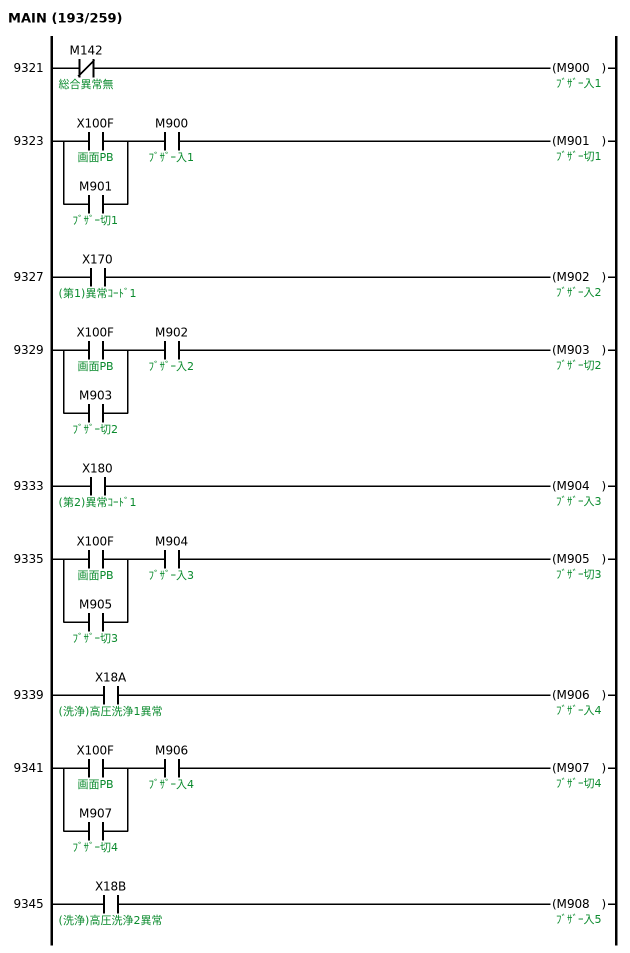
[picture p192: ladder of MAIN, rungs at steps 9321 to 9345]
9321  LDI     M142  ; 総合異常無
      OUT     M900  ; ﾌﾞｻﾞｰ入1
9323  LD      X100F  ; 画面PB
      OR      M901  ; ﾌﾞｻﾞｰ切1
      AND     M900  ; ﾌﾞｻﾞｰ入1
      OUT     M901  ; ﾌﾞｻﾞｰ切1
9327  LD      X170  ; (第1)異常ｺｰﾄﾞ1
      OUT     M902  ; ﾌﾞｻﾞｰ入2
9329  LD      X100F  ; 画面PB
      OR      M903  ; ﾌﾞｻﾞｰ切2
      AND     M902  ; ﾌﾞｻﾞｰ入2
      OUT     M903  ; ﾌﾞｻﾞｰ切2
9333  LD      X180  ; (第2)異常ｺｰﾄﾞ1
      OUT     M904  ; ﾌﾞｻﾞｰ入3
9335  LD      X100F  ; 画面PB
      OR      M905  ; ﾌﾞｻﾞｰ切3
      AND     M904  ; ﾌﾞｻﾞｰ入3
      OUT     M905  ; ﾌﾞｻﾞｰ切3
9339  LD      X18A  ; (洗浄)高圧洗浄1異常
      OUT     M906  ; ﾌﾞｻﾞｰ入4
9341  LD      X100F  ; 画面PB
      OR      M907  ; ﾌﾞｻﾞｰ切4
      AND     M906  ; ﾌﾞｻﾞｰ入4
      OUT     M907  ; ﾌﾞｻﾞｰ切4
9345  LD      X18B  ; (洗浄)高圧洗浄2異常
      OUT     M908  ; ﾌﾞｻﾞｰ入5
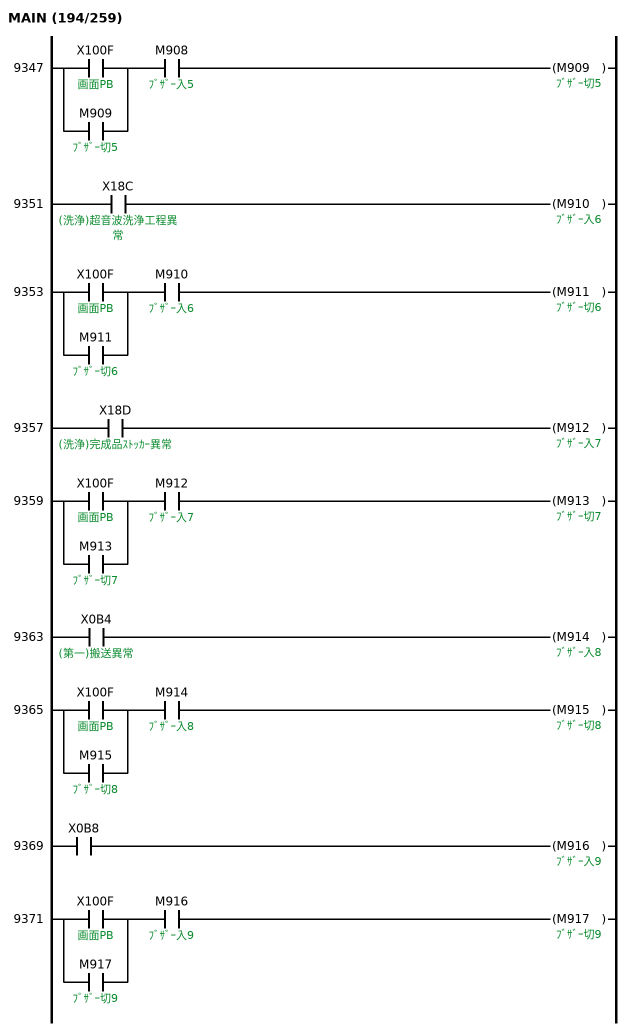
9347  LD      X100F  ; 画面PB
      OR      M909  ; ﾌﾞｻﾞｰ切5
      AND     M908  ; ﾌﾞｻﾞｰ入5
      OUT     M909  ; ﾌﾞｻﾞｰ切5
9351  LD      X18C  ; (洗浄)超音波洗浄工程異常
      OUT     M910  ; ﾌﾞｻﾞｰ入6
9353  LD      X100F  ; 画面PB
      OR      M911  ; ﾌﾞｻﾞｰ切6
      AND     M910  ; ﾌﾞｻﾞｰ入6
      OUT     M911  ; ﾌﾞｻﾞｰ切6
9357  LD      X18D  ; (洗浄)完成品ｽﾄｯｶｰ異常
      OUT     M912  ; ﾌﾞｻﾞｰ入7
9359  LD      X100F  ; 画面PB
      OR      M913  ; ﾌﾞｻﾞｰ切7
      AND     M912  ; ﾌﾞｻﾞｰ入7
      OUT     M913  ; ﾌﾞｻﾞｰ切7
9363  LD      X0B4  ; (第一)搬送異常
      OUT     M914  ; ﾌﾞｻﾞｰ入8
9365  LD      X100F  ; 画面PB
      OR      M915  ; ﾌﾞｻﾞｰ切8
      AND     M914  ; ﾌﾞｻﾞｰ入8
      OUT     M915  ; ﾌﾞｻﾞｰ切8
9369  LD      X0B8
      OUT     M916  ; ﾌﾞｻﾞｰ入9
9371  LD      X100F  ; 画面PB
      OR      M917  ; ﾌﾞｻﾞｰ切9
      AND     M916  ; ﾌﾞｻﾞｰ入9
      OUT     M917  ; ﾌﾞｻﾞｰ切9
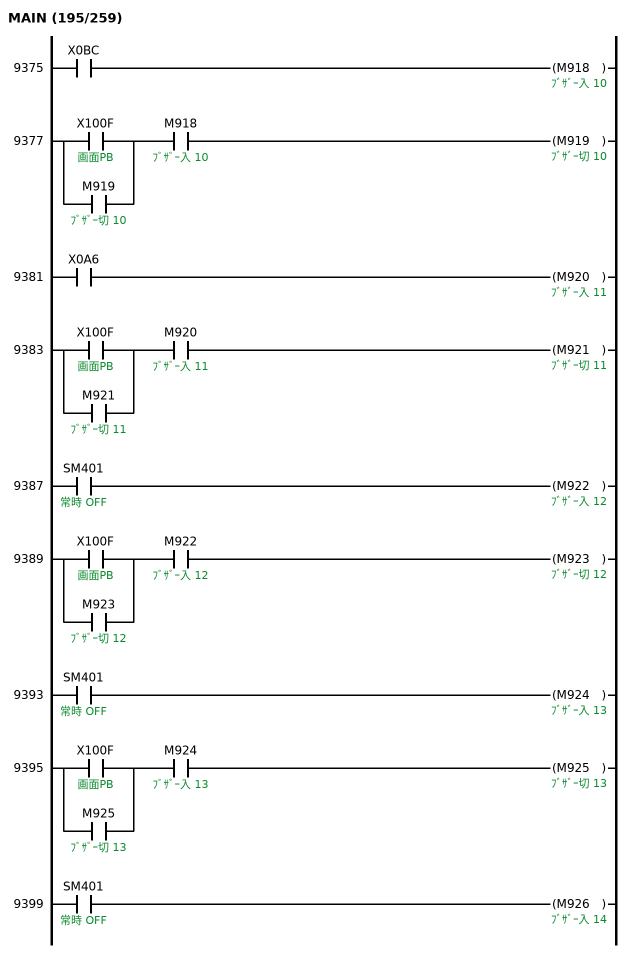
9375  LD      X0BC
      OUT     M918  ; ﾌﾞｻﾞｰ入 10
9377  LD      X100F  ; 画面PB
      OR      M919  ; ﾌﾞｻﾞｰ切 10
      AND     M918  ; ﾌﾞｻﾞｰ入 10
      OUT     M919  ; ﾌﾞｻﾞｰ切 10
9381  LD      X0A6
      OUT     M920  ; ﾌﾞｻﾞｰ入 11
9383  LD      X100F  ; 画面PB
      OR      M921  ; ﾌﾞｻﾞｰ切 11
      AND     M920  ; ﾌﾞｻﾞｰ入 11
      OUT     M921  ; ﾌﾞｻﾞｰ切 11
9387  LD      SM401  ; 常時 OFF
      OUT     M922  ; ﾌﾞｻﾞｰ入 12
9389  LD      X100F  ; 画面PB
      OR      M923  ; ﾌﾞｻﾞｰ切 12
      AND     M922  ; ﾌﾞｻﾞｰ入 12
      OUT     M923  ; ﾌﾞｻﾞｰ切 12
9393  LD      SM401  ; 常時 OFF
      OUT     M924  ; ﾌﾞｻﾞｰ入 13
9395  LD      X100F  ; 画面PB
      OR      M925  ; ﾌﾞｻﾞｰ切 13
      AND     M924  ; ﾌﾞｻﾞｰ入 13
      OUT     M925  ; ﾌﾞｻﾞｰ切 13
9399  LD      SM401  ; 常時 OFF
      OUT     M926  ; ﾌﾞｻﾞｰ入 14
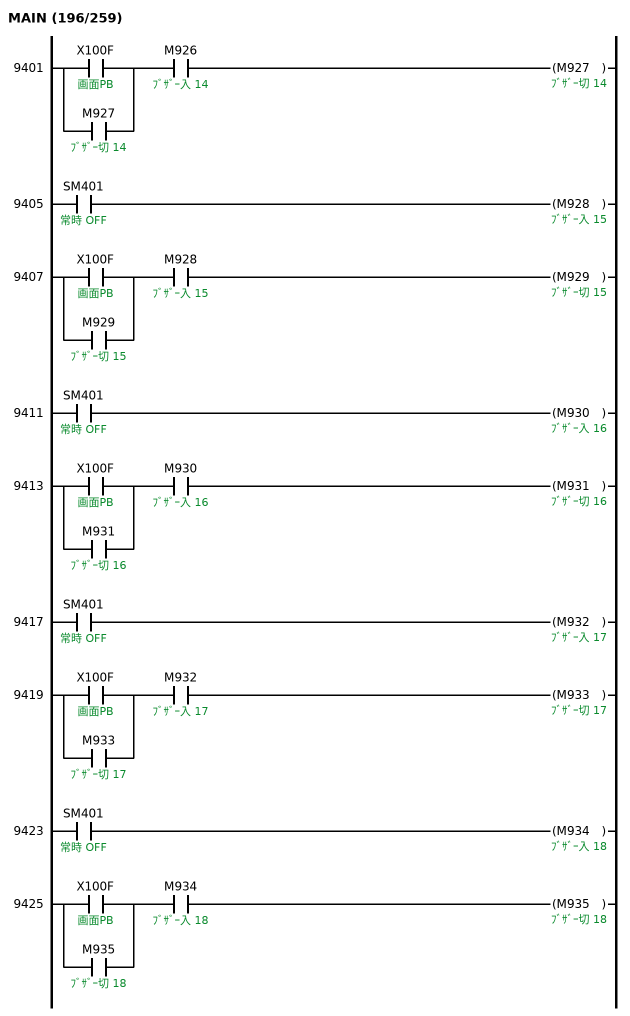
9401  LD      X100F  ; 画面PB
      OR      M927  ; ﾌﾞｻﾞｰ切 14
      AND     M926  ; ﾌﾞｻﾞｰ入 14
      OUT     M927  ; ﾌﾞｻﾞｰ切 14
9405  LD      SM401  ; 常時 OFF
      OUT     M928  ; ﾌﾞｻﾞｰ入 15
9407  LD      X100F  ; 画面PB
      OR      M929  ; ﾌﾞｻﾞｰ切 15
      AND     M928  ; ﾌﾞｻﾞｰ入 15
      OUT     M929  ; ﾌﾞｻﾞｰ切 15
9411  LD      SM401  ; 常時 OFF
      OUT     M930  ; ﾌﾞｻﾞｰ入 16
9413  LD      X100F  ; 画面PB
      OR      M931  ; ﾌﾞｻﾞｰ切 16
      AND     M930  ; ﾌﾞｻﾞｰ入 16
      OUT     M931  ; ﾌﾞｻﾞｰ切 16
9417  LD      SM401  ; 常時 OFF
      OUT     M932  ; ﾌﾞｻﾞｰ入 17
9419  LD      X100F  ; 画面PB
      OR      M933  ; ﾌﾞｻﾞｰ切 17
      AND     M932  ; ﾌﾞｻﾞｰ入 17
      OUT     M933  ; ﾌﾞｻﾞｰ切 17
9423  LD      SM401  ; 常時 OFF
      OUT     M934  ; ﾌﾞｻﾞｰ入 18
9425  LD      X100F  ; 画面PB
      OR      M935  ; ﾌﾞｻﾞｰ切 18
      AND     M934  ; ﾌﾞｻﾞｰ入 18
      OUT     M935  ; ﾌﾞｻﾞｰ切 18
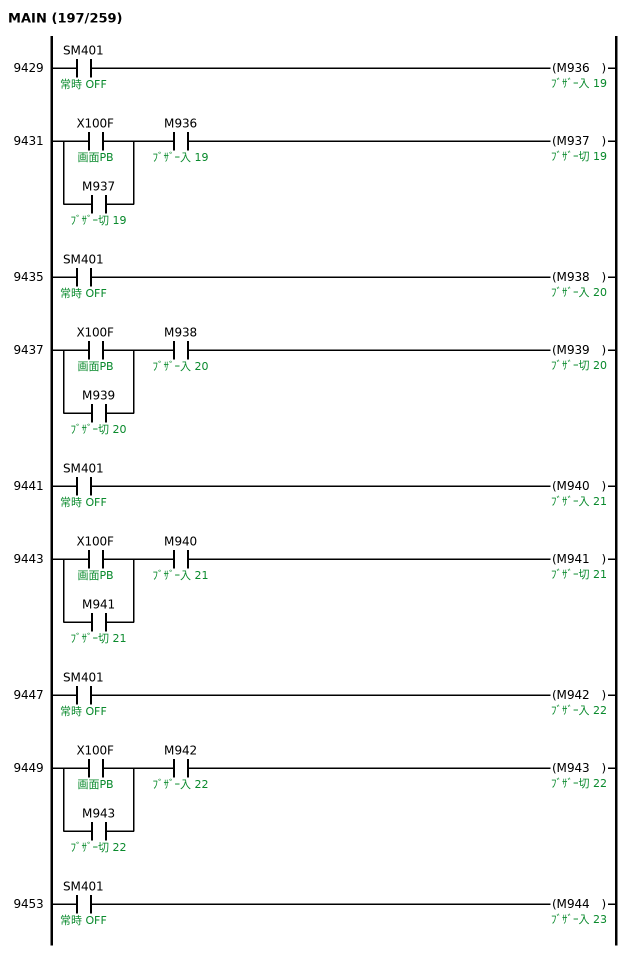
9429  LD      SM401  ; 常時 OFF
      OUT     M936  ; ﾌﾞｻﾞｰ入 19
9431  LD      X100F  ; 画面PB
      OR      M937  ; ﾌﾞｻﾞｰ切 19
      AND     M936  ; ﾌﾞｻﾞｰ入 19
      OUT     M937  ; ﾌﾞｻﾞｰ切 19
9435  LD      SM401  ; 常時 OFF
      OUT     M938  ; ﾌﾞｻﾞｰ入 20
9437  LD      X100F  ; 画面PB
      OR      M939  ; ﾌﾞｻﾞｰ切 20
      AND     M938  ; ﾌﾞｻﾞｰ入 20
      OUT     M939  ; ﾌﾞｻﾞｰ切 20
9441  LD      SM401  ; 常時 OFF
      OUT     M940  ; ﾌﾞｻﾞｰ入 21
9443  LD      X100F  ; 画面PB
      OR      M941  ; ﾌﾞｻﾞｰ切 21
      AND     M940  ; ﾌﾞｻﾞｰ入 21
      OUT     M941  ; ﾌﾞｻﾞｰ切 21
9447  LD      SM401  ; 常時 OFF
      OUT     M942  ; ﾌﾞｻﾞｰ入 22
9449  LD      X100F  ; 画面PB
      OR      M943  ; ﾌﾞｻﾞｰ切 22
      AND     M942  ; ﾌﾞｻﾞｰ入 22
      OUT     M943  ; ﾌﾞｻﾞｰ切 22
9453  LD      SM401  ; 常時 OFF
      OUT     M944  ; ﾌﾞｻﾞｰ入 23
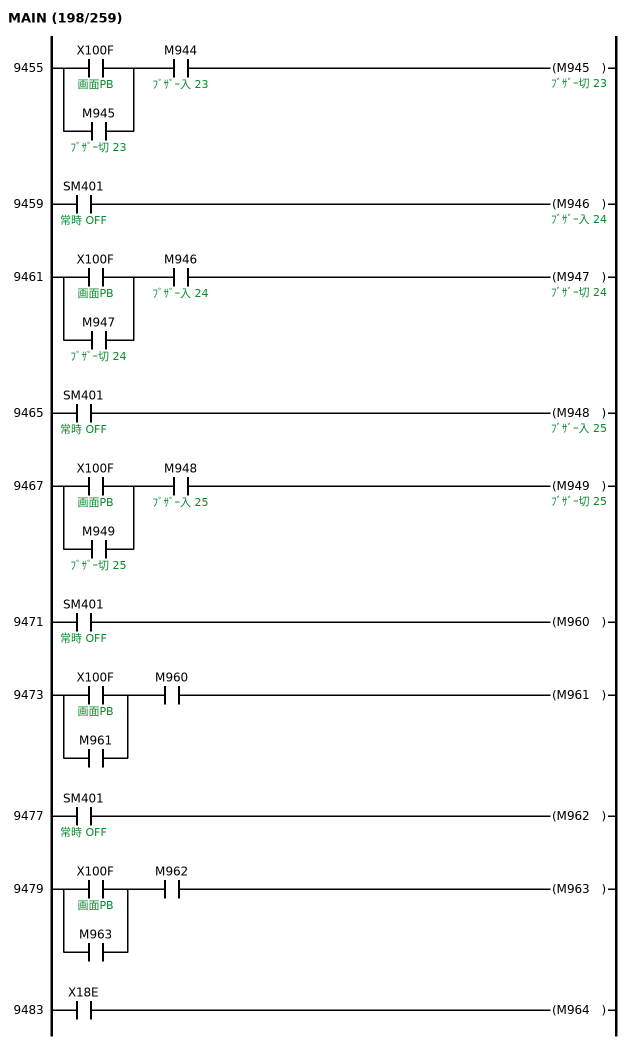
9455  LD      X100F  ; 画面PB
      OR      M945  ; ﾌﾞｻﾞｰ切 23
      AND     M944  ; ﾌﾞｻﾞｰ入 23
      OUT     M945  ; ﾌﾞｻﾞｰ切 23
9459  LD      SM401  ; 常時 OFF
      OUT     M946  ; ﾌﾞｻﾞｰ入 24
9461  LD      X100F  ; 画面PB
      OR      M947  ; ﾌﾞｻﾞｰ切 24
      AND     M946  ; ﾌﾞｻﾞｰ入 24
      OUT     M947  ; ﾌﾞｻﾞｰ切 24
9465  LD      SM401  ; 常時 OFF
      OUT     M948  ; ﾌﾞｻﾞｰ入 25
9467  LD      X100F  ; 画面PB
      OR      M949  ; ﾌﾞｻﾞｰ切 25
      AND     M948  ; ﾌﾞｻﾞｰ入 25
      OUT     M949  ; ﾌﾞｻﾞｰ切 25
9471  LD      SM401  ; 常時 OFF
      OUT     M960
9473  LD      X100F  ; 画面PB
      OR      M961
      AND     M960
      OUT     M961
9477  LD      SM401  ; 常時 OFF
      OUT     M962
9479  LD      X100F  ; 画面PB
      OR      M963
      AND     M962
      OUT     M963
9483  LD      X18E
      OUT     M964
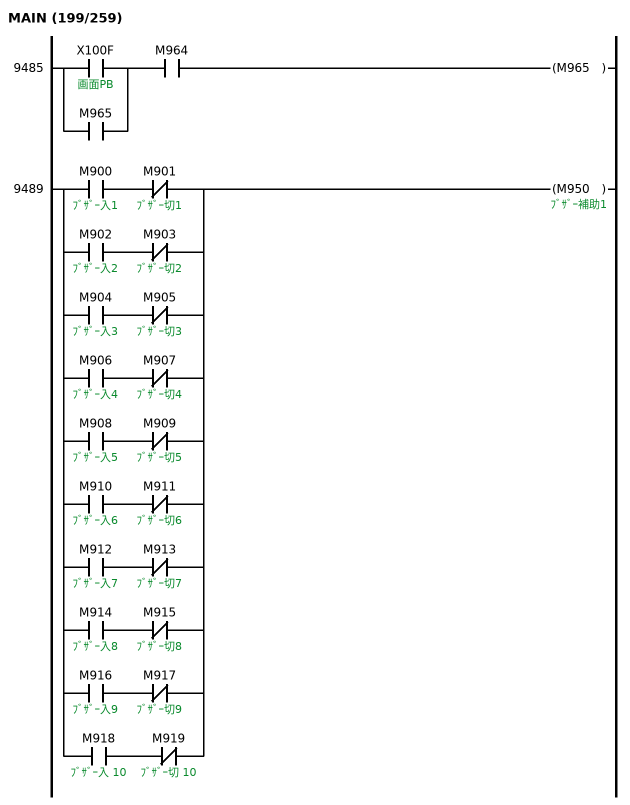
9485  LD      X100F  ; 画面PB
      OR      M965
      AND     M964
      OUT     M965
9489  LD      M900  ; ﾌﾞｻﾞｰ入1
      ANI     M901  ; ﾌﾞｻﾞｰ切1
      LD      M902  ; ﾌﾞｻﾞｰ入2
      ANI     M903  ; ﾌﾞｻﾞｰ切2
      ORB
      LD      M904  ; ﾌﾞｻﾞｰ入3
      ANI     M905  ; ﾌﾞｻﾞｰ切3
      ORB
      LD      M906  ; ﾌﾞｻﾞｰ入4
      ANI     M907  ; ﾌﾞｻﾞｰ切4
      ORB
      LD      M908  ; ﾌﾞｻﾞｰ入5
      ANI     M909  ; ﾌﾞｻﾞｰ切5
      ORB
      LD      M910  ; ﾌﾞｻﾞｰ入6
      ANI     M911  ; ﾌﾞｻﾞｰ切6
      ORB
      LD      M912  ; ﾌﾞｻﾞｰ入7
      ANI     M913  ; ﾌﾞｻﾞｰ切7
      ORB
      LD      M914  ; ﾌﾞｻﾞｰ入8
      ANI     M915  ; ﾌﾞｻﾞｰ切8
      ORB
      LD      M916  ; ﾌﾞｻﾞｰ入9
      ANI     M917  ; ﾌﾞｻﾞｰ切9
      ORB
      LD      M918  ; ﾌﾞｻﾞｰ入 10
      ANI     M919  ; ﾌﾞｻﾞｰ切 10
      ORB
      OUT     M950  ; ﾌﾞｻﾞｰ補助1
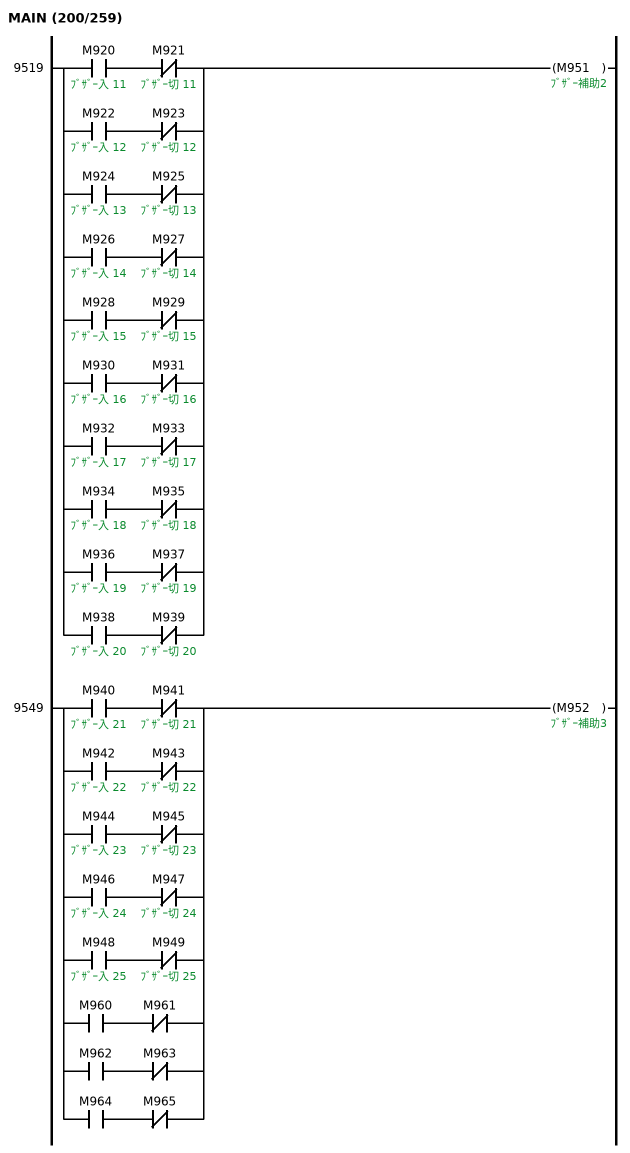
9519  LD      M920  ; ﾌﾞｻﾞｰ入 11
      ANI     M921  ; ﾌﾞｻﾞｰ切 11
      LD      M922  ; ﾌﾞｻﾞｰ入 12
      ANI     M923  ; ﾌﾞｻﾞｰ切 12
      ORB
      LD      M924  ; ﾌﾞｻﾞｰ入 13
      ANI     M925  ; ﾌﾞｻﾞｰ切 13
      ORB
      LD      M926  ; ﾌﾞｻﾞｰ入 14
      ANI     M927  ; ﾌﾞｻﾞｰ切 14
      ORB
      LD      M928  ; ﾌﾞｻﾞｰ入 15
      ANI     M929  ; ﾌﾞｻﾞｰ切 15
      ORB
      LD      M930  ; ﾌﾞｻﾞｰ入 16
      ANI     M931  ; ﾌﾞｻﾞｰ切 16
      ORB
      LD      M932  ; ﾌﾞｻﾞｰ入 17
      ANI     M933  ; ﾌﾞｻﾞｰ切 17
      ORB
      LD      M934  ; ﾌﾞｻﾞｰ入 18
      ANI     M935  ; ﾌﾞｻﾞｰ切 18
      ORB
      LD      M936  ; ﾌﾞｻﾞｰ入 19
      ANI     M937  ; ﾌﾞｻﾞｰ切 19
      ORB
      LD      M938  ; ﾌﾞｻﾞｰ入 20
      ANI     M939  ; ﾌﾞｻﾞｰ切 20
      ORB
      OUT     M951  ; ﾌﾞｻﾞｰ補助2
9549  LD      M940  ; ﾌﾞｻﾞｰ入 21
      ANI     M941  ; ﾌﾞｻﾞｰ切 21
      LD      M942  ; ﾌﾞｻﾞｰ入 22
      ANI     M943  ; ﾌﾞｻﾞｰ切 22
      ORB
      LD      M944  ; ﾌﾞｻﾞｰ入 23
      ANI     M945  ; ﾌﾞｻﾞｰ切 23
      ORB
      LD      M946  ; ﾌﾞｻﾞｰ入 24
      ANI     M947  ; ﾌﾞｻﾞｰ切 24
      ORB
      LD      M948  ; ﾌﾞｻﾞｰ入 25
      ANI     M949  ; ﾌﾞｻﾞｰ切 25
      ORB
      LD      M960
      ANI     M961
      ORB
      LD      M962
      ANI     M963
      ORB
      LD      M964
      ANI     M965
      ORB
      OUT     M952  ; ﾌﾞｻﾞｰ補助3
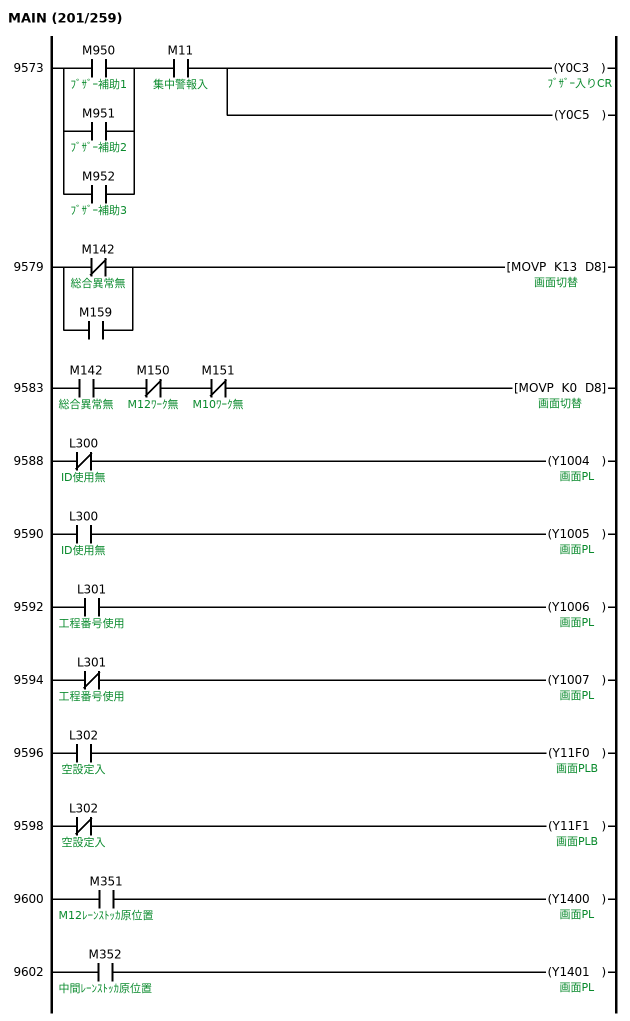
9573  LD      M950  ; ﾌﾞｻﾞｰ補助1
      OR      M951  ; ﾌﾞｻﾞｰ補助2
      OR      M952  ; ﾌﾞｻﾞｰ補助3
      AND     M11  ; 集中警報入
      OUT     Y0C3  ; ﾌﾞｻﾞｰ入りCR
      OUT     Y0C5
9579  LDI     M142  ; 総合異常無
      OR      M159
      MOVP    K13 D8  ; 画面切替
9583  LD      M142  ; 総合異常無
      ANI     M150  ; M12ﾜｰｸ無
      ANI     M151  ; M10ﾜｰｸ無
      MOVP    K0 D8
9588  LDI     L300  ; ID使用無
      OUT     Y1004  ; 画面PL
9590  LD      L300  ; ID使用無
      OUT     Y1005  ; 画面PL
9592  LD      L301  ; 工程番号使用
      OUT     Y1006  ; 画面PL
9594  LDI     L301  ; 工程番号使用
      OUT     Y1007  ; 画面PL
9596  LD      L302  ; 空設定入
      OUT     Y11F0  ; 画面PLB
9598  LDI     L302  ; 空設定入
      OUT     Y11F1  ; 画面PLB
9600  LD      M351  ; M12ﾚｰﾝｽﾄｯｶ原位置
      OUT     Y1400  ; 画面PL
9602  LD      M352  ; 中間ﾚｰﾝｽﾄｯｶ原位置
      OUT     Y1401  ; 画面PL
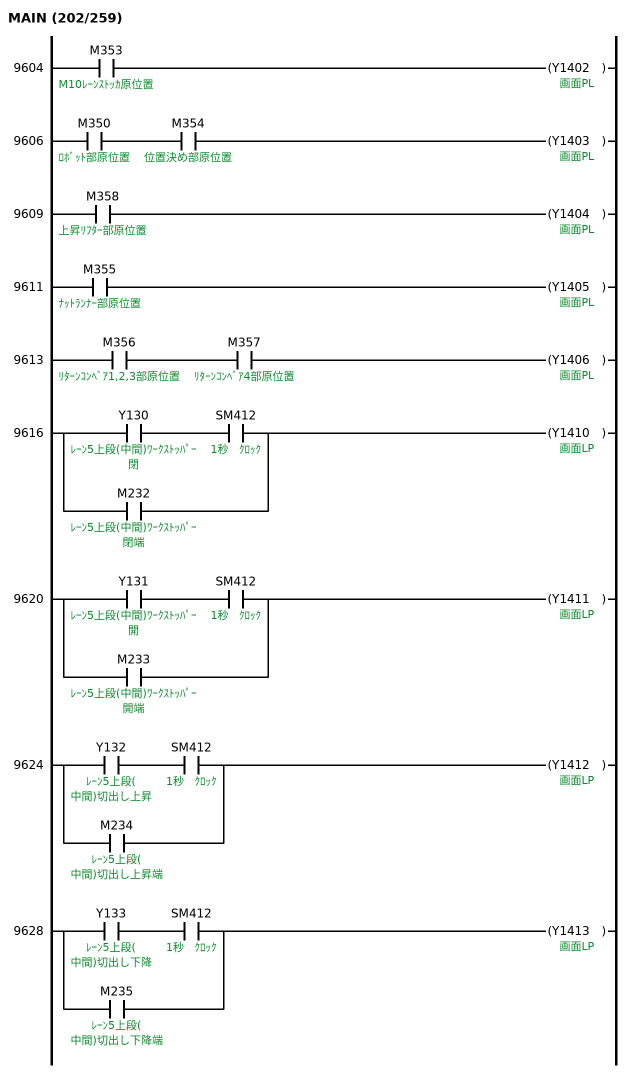
9604  LD      M353  ; M10ﾚｰﾝｽﾄｯｶ原位置
      OUT     Y1402  ; 画面PL
9606  LD      M350  ; ﾛﾎﾞｯﾄ部原位置
      AND     M354  ; 位置決め部原位置
      OUT     Y1403  ; 画面PL
9609  LD      M358  ; 上昇ﾘﾌﾀｰ部原位置
      OUT     Y1404  ; 画面PL
9611  LD      M355  ; ﾅｯﾄﾗﾝﾅｰ部原位置
      OUT     Y1405  ; 画面PL
9613  LD      M356  ; ﾘﾀｰﾝｺﾝﾍﾞｱ1,2,3部原位置
      AND     M357  ; ﾘﾀｰﾝｺﾝﾍﾞｱ4部原位置
      OUT     Y1406  ; 画面PL
9616  LD      Y130  ; ﾚｰﾝ5上段(中間)ﾜｰｸｽﾄｯﾊﾟｰ閉
      AND     SM412  ; 1秒   ｸﾛｯｸ
      OR      M232  ; ﾚｰﾝ5上段(中間)ﾜｰｸｽﾄｯﾊﾟｰ閉端
      OUT     Y1410  ; 画面LP
9620  LD      Y131  ; ﾚｰﾝ5上段(中間)ﾜｰｸｽﾄｯﾊﾟｰ開
      AND     SM412  ; 1秒   ｸﾛｯｸ
      OR      M233  ; ﾚｰﾝ5上段(中間)ﾜｰｸｽﾄｯﾊﾟｰ開端
      OUT     Y1411  ; 画面LP
9624  LD      Y132  ; ﾚｰﾝ5上段(中間)切出し上昇
      AND     SM412  ; 1秒   ｸﾛｯｸ
      OR      M234  ; ﾚｰﾝ5上段(中間)切出し上昇端
      OUT     Y1412  ; 画面LP
9628  LD      Y133  ; ﾚｰﾝ5上段(中間)切出し下降
      AND     SM412  ; 1秒   ｸﾛｯｸ
      OR      M235  ; ﾚｰﾝ5上段(中間)切出し下降端
      OUT     Y1413  ; 画面LP
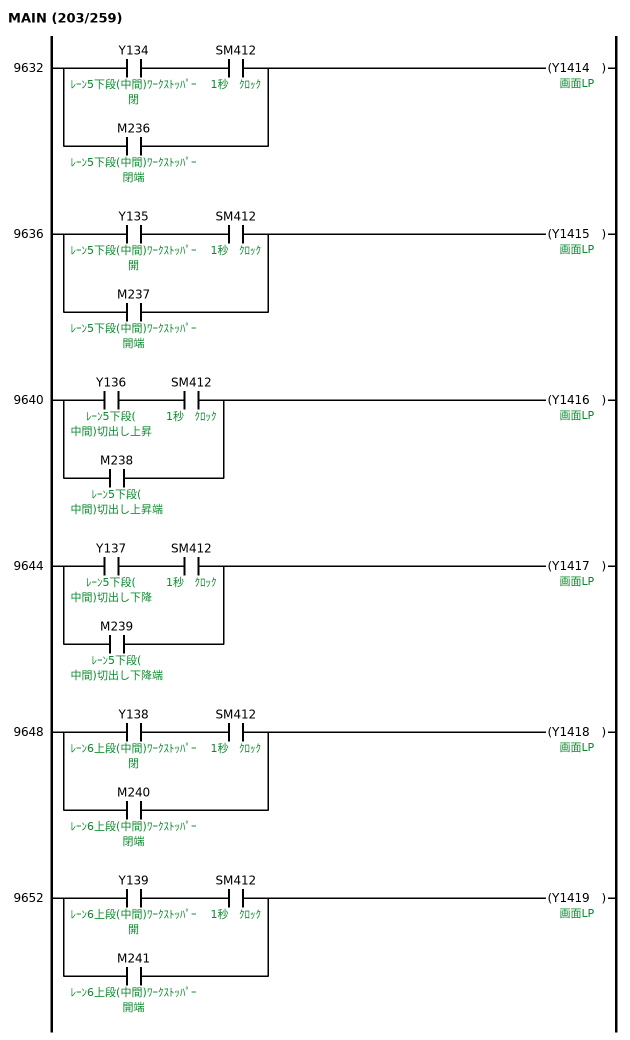
9632  LD      Y134  ; ﾚｰﾝ5下段(中間)ﾜｰｸｽﾄｯﾊﾟｰ閉
      AND     SM412  ; 1秒   ｸﾛｯｸ
      OR      M236  ; ﾚｰﾝ5下段(中間)ﾜｰｸｽﾄｯﾊﾟｰ閉端
      OUT     Y1414  ; 画面LP
9636  LD      Y135  ; ﾚｰﾝ5下段(中間)ﾜｰｸｽﾄｯﾊﾟｰ開
      AND     SM412  ; 1秒   ｸﾛｯｸ
      OR      M237  ; ﾚｰﾝ5下段(中間)ﾜｰｸｽﾄｯﾊﾟｰ開端
      OUT     Y1415  ; 画面LP
9640  LD      Y136  ; ﾚｰﾝ5下段(中間)切出し上昇
      AND     SM412  ; 1秒   ｸﾛｯｸ
      OR      M238  ; ﾚｰﾝ5下段(中間)切出し上昇端
      OUT     Y1416  ; 画面LP
9644  LD      Y137  ; ﾚｰﾝ5下段(中間)切出し下降
      AND     SM412  ; 1秒   ｸﾛｯｸ
      OR      M239  ; ﾚｰﾝ5下段(中間)切出し下降端
      OUT     Y1417  ; 画面LP
9648  LD      Y138  ; ﾚｰﾝ6上段(中間)ﾜｰｸｽﾄｯﾊﾟｰ閉
      AND     SM412  ; 1秒   ｸﾛｯｸ
      OR      M240  ; ﾚｰﾝ6上段(中間)ﾜｰｸｽﾄｯﾊﾟｰ閉端
      OUT     Y1418  ; 画面LP
9652  LD      Y139  ; ﾚｰﾝ6上段(中間)ﾜｰｸｽﾄｯﾊﾟｰ開
      AND     SM412  ; 1秒   ｸﾛｯｸ
      OR      M241  ; ﾚｰﾝ6上段(中間)ﾜｰｸｽﾄｯﾊﾟｰ開端
      OUT     Y1419  ; 画面LP
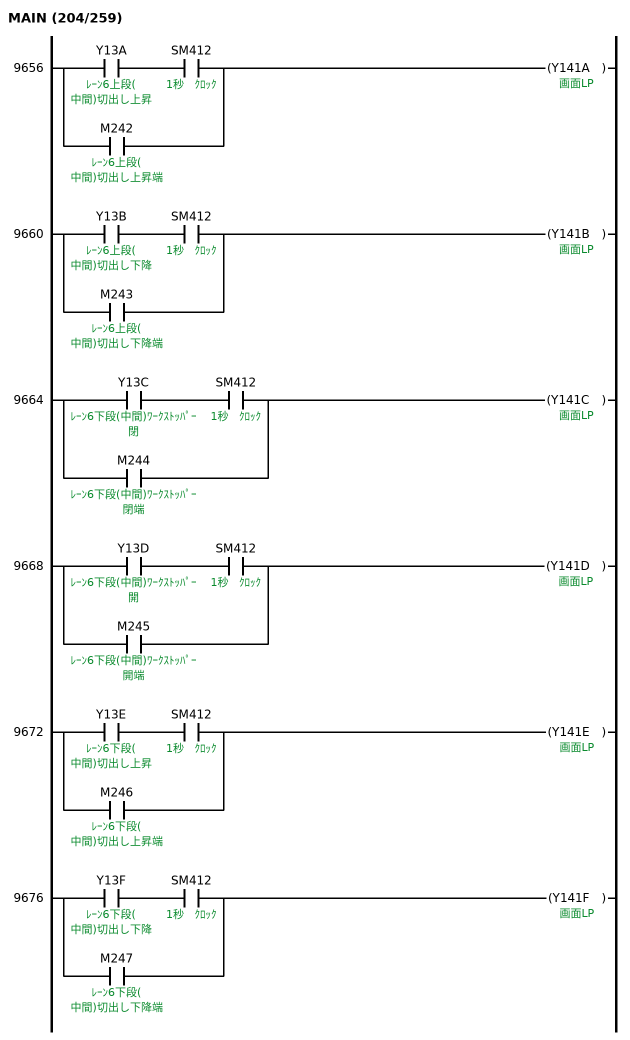
9656  LD      Y13A  ; ﾚｰﾝ6上段(中間)切出し上昇
      AND     SM412  ; 1秒   ｸﾛｯｸ
      OR      M242  ; ﾚｰﾝ6上段(中間)切出し上昇端
      OUT     Y141A  ; 画面LP
9660  LD      Y13B  ; ﾚｰﾝ6上段(中間)切出し下降
      AND     SM412  ; 1秒   ｸﾛｯｸ
      OR      M243  ; ﾚｰﾝ6上段(中間)切出し下降端
      OUT     Y141B  ; 画面LP
9664  LD      Y13C  ; ﾚｰﾝ6下段(中間)ﾜｰｸｽﾄｯﾊﾟｰ閉
      AND     SM412  ; 1秒   ｸﾛｯｸ
      OR      M244  ; ﾚｰﾝ6下段(中間)ﾜｰｸｽﾄｯﾊﾟｰ閉端
      OUT     Y141C  ; 画面LP
9668  LD      Y13D  ; ﾚｰﾝ6下段(中間)ﾜｰｸｽﾄｯﾊﾟｰ開
      AND     SM412  ; 1秒   ｸﾛｯｸ
      OR      M245  ; ﾚｰﾝ6下段(中間)ﾜｰｸｽﾄｯﾊﾟｰ開端
      OUT     Y141D  ; 画面LP
9672  LD      Y13E  ; ﾚｰﾝ6下段(中間)切出し上昇
      AND     SM412  ; 1秒   ｸﾛｯｸ
      OR      M246  ; ﾚｰﾝ6下段(中間)切出し上昇端
      OUT     Y141E  ; 画面LP
9676  LD      Y13F  ; ﾚｰﾝ6下段(中間)切出し下降
      AND     SM412  ; 1秒   ｸﾛｯｸ
      OR      M247  ; ﾚｰﾝ6下段(中間)切出し下降端
      OUT     Y141F  ; 画面LP
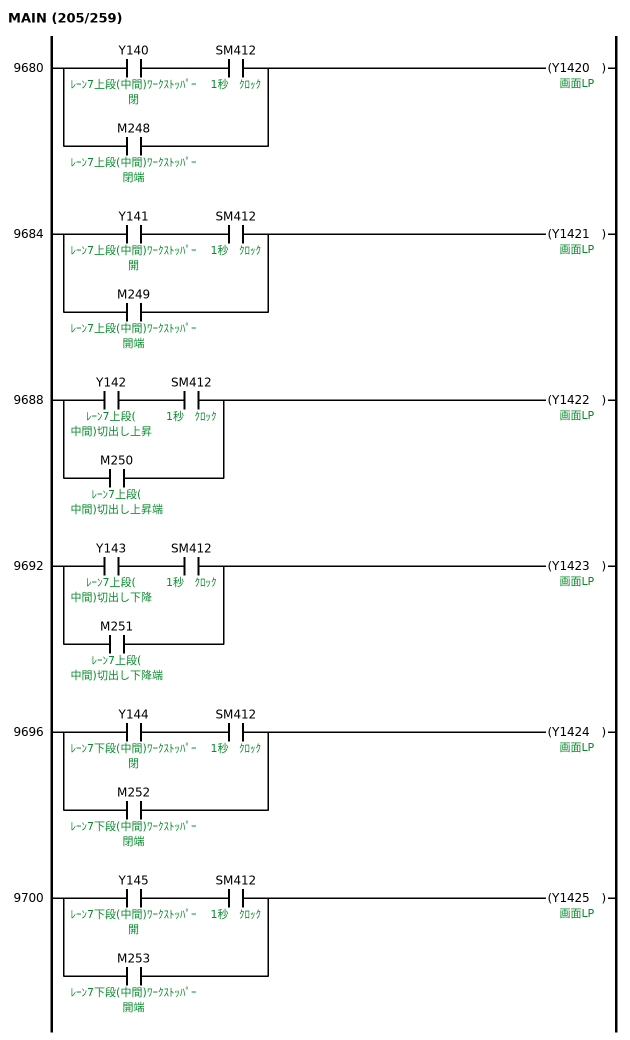
9680  LD      Y140  ; ﾚｰﾝ7上段(中間)ﾜｰｸｽﾄｯﾊﾟｰ閉
      AND     SM412  ; 1秒   ｸﾛｯｸ
      OR      M248  ; ﾚｰﾝ7上段(中間)ﾜｰｸｽﾄｯﾊﾟｰ閉端
      OUT     Y1420  ; 画面LP
9684  LD      Y141  ; ﾚｰﾝ7上段(中間)ﾜｰｸｽﾄｯﾊﾟｰ開
      AND     SM412  ; 1秒   ｸﾛｯｸ
      OR      M249  ; ﾚｰﾝ7上段(中間)ﾜｰｸｽﾄｯﾊﾟｰ開端
      OUT     Y1421  ; 画面LP
9688  LD      Y142  ; ﾚｰﾝ7上段(中間)切出し上昇
      AND     SM412  ; 1秒   ｸﾛｯｸ
      OR      M250  ; ﾚｰﾝ7上段(中間)切出し上昇端
      OUT     Y1422  ; 画面LP
9692  LD      Y143  ; ﾚｰﾝ7上段(中間)切出し下降
      AND     SM412  ; 1秒   ｸﾛｯｸ
      OR      M251  ; ﾚｰﾝ7上段(中間)切出し下降端
      OUT     Y1423  ; 画面LP
9696  LD      Y144  ; ﾚｰﾝ7下段(中間)ﾜｰｸｽﾄｯﾊﾟｰ閉
      AND     SM412  ; 1秒   ｸﾛｯｸ
      OR      M252  ; ﾚｰﾝ7下段(中間)ﾜｰｸｽﾄｯﾊﾟｰ閉端
      OUT     Y1424  ; 画面LP
9700  LD      Y145  ; ﾚｰﾝ7下段(中間)ﾜｰｸｽﾄｯﾊﾟｰ開
      AND     SM412  ; 1秒   ｸﾛｯｸ
      OR      M253  ; ﾚｰﾝ7下段(中間)ﾜｰｸｽﾄｯﾊﾟｰ開端
      OUT     Y1425  ; 画面LP
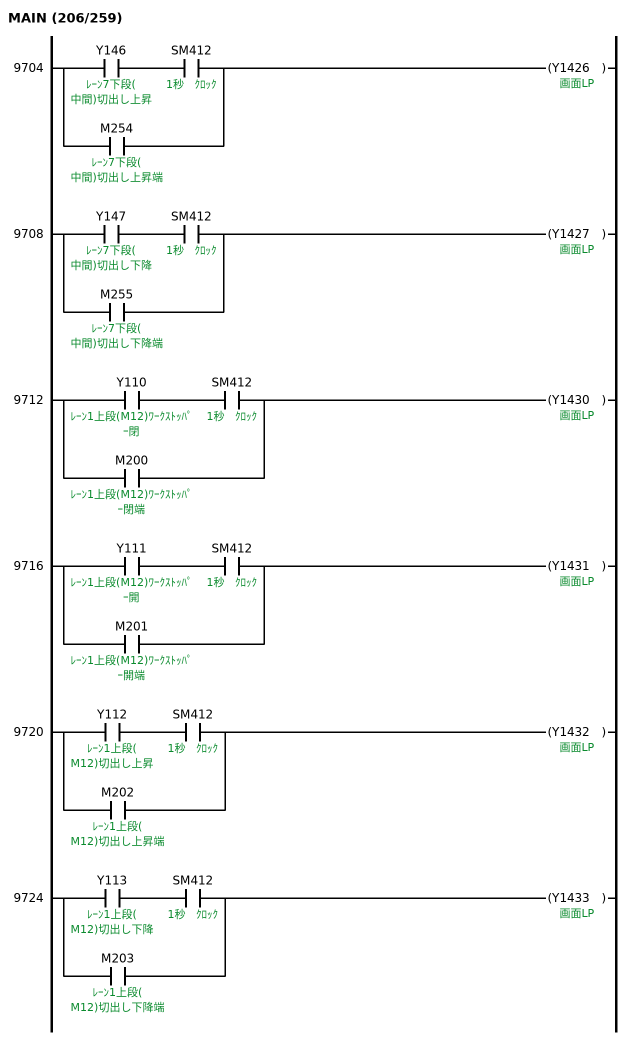
9704  LD      Y146  ; ﾚｰﾝ7下段(中間)切出し上昇
      AND     SM412  ; 1秒   ｸﾛｯｸ
      OR      M254  ; ﾚｰﾝ7下段(中間)切出し上昇端
      OUT     Y1426  ; 画面LP
9708  LD      Y147  ; ﾚｰﾝ7下段(中間)切出し下降
      AND     SM412  ; 1秒   ｸﾛｯｸ
      OR      M255  ; ﾚｰﾝ7下段(中間)切出し下降端
      OUT     Y1427  ; 画面LP
9712  LD      Y110  ; ﾚｰﾝ1上段(M12)ﾜｰｸｽﾄｯﾊﾟｰ閉
      AND     SM412  ; 1秒   ｸﾛｯｸ
      OR      M200  ; ﾚｰﾝ1上段(M12)ﾜｰｸｽﾄｯﾊﾟｰ閉端
      OUT     Y1430  ; 画面LP
9716  LD      Y111  ; ﾚｰﾝ1上段(M12)ﾜｰｸｽﾄｯﾊﾟｰ開
      AND     SM412  ; 1秒   ｸﾛｯｸ
      OR      M201  ; ﾚｰﾝ1上段(M12)ﾜｰｸｽﾄｯﾊﾟｰ開端
      OUT     Y1431  ; 画面LP
9720  LD      Y112  ; ﾚｰﾝ1上段(M12)切出し上昇
      AND     SM412  ; 1秒   ｸﾛｯｸ
      OR      M202  ; ﾚｰﾝ1上段(M12)切出し上昇端
      OUT     Y1432  ; 画面LP
9724  LD      Y113  ; ﾚｰﾝ1上段(M12)切出し下降
      AND     SM412  ; 1秒   ｸﾛｯｸ
      OR      M203  ; ﾚｰﾝ1上段(M12)切出し下降端
      OUT     Y1433  ; 画面LP
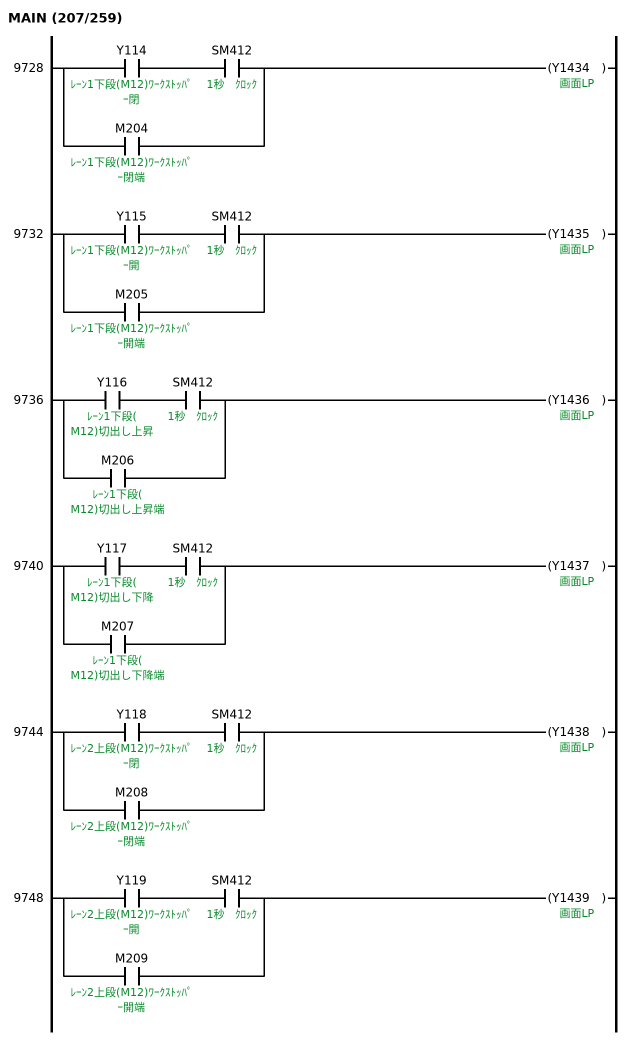
9728  LD      Y114  ; ﾚｰﾝ1下段(M12)ﾜｰｸｽﾄｯﾊﾟｰ閉
      AND     SM412  ; 1秒   ｸﾛｯｸ
      OR      M204  ; ﾚｰﾝ1下段(M12)ﾜｰｸｽﾄｯﾊﾟｰ閉端
      OUT     Y1434  ; 画面LP
9732  LD      Y115  ; ﾚｰﾝ1下段(M12)ﾜｰｸｽﾄｯﾊﾟｰ開
      AND     SM412  ; 1秒   ｸﾛｯｸ
      OR      M205  ; ﾚｰﾝ1下段(M12)ﾜｰｸｽﾄｯﾊﾟｰ開端
      OUT     Y1435  ; 画面LP
9736  LD      Y116  ; ﾚｰﾝ1下段(M12)切出し上昇
      AND     SM412  ; 1秒   ｸﾛｯｸ
      OR      M206  ; ﾚｰﾝ1下段(M12)切出し上昇端
      OUT     Y1436  ; 画面LP
9740  LD      Y117  ; ﾚｰﾝ1下段(M12)切出し下降
      AND     SM412  ; 1秒   ｸﾛｯｸ
      OR      M207  ; ﾚｰﾝ1下段(M12)切出し下降端
      OUT     Y1437  ; 画面LP
9744  LD      Y118  ; ﾚｰﾝ2上段(M12)ﾜｰｸｽﾄｯﾊﾟｰ閉
      AND     SM412  ; 1秒   ｸﾛｯｸ
      OR      M208  ; ﾚｰﾝ2上段(M12)ﾜｰｸｽﾄｯﾊﾟｰ閉端
      OUT     Y1438  ; 画面LP
9748  LD      Y119  ; ﾚｰﾝ2上段(M12)ﾜｰｸｽﾄｯﾊﾟｰ開
      AND     SM412  ; 1秒   ｸﾛｯｸ
      OR      M209  ; ﾚｰﾝ2上段(M12)ﾜｰｸｽﾄｯﾊﾟｰ開端
      OUT     Y1439  ; 画面LP
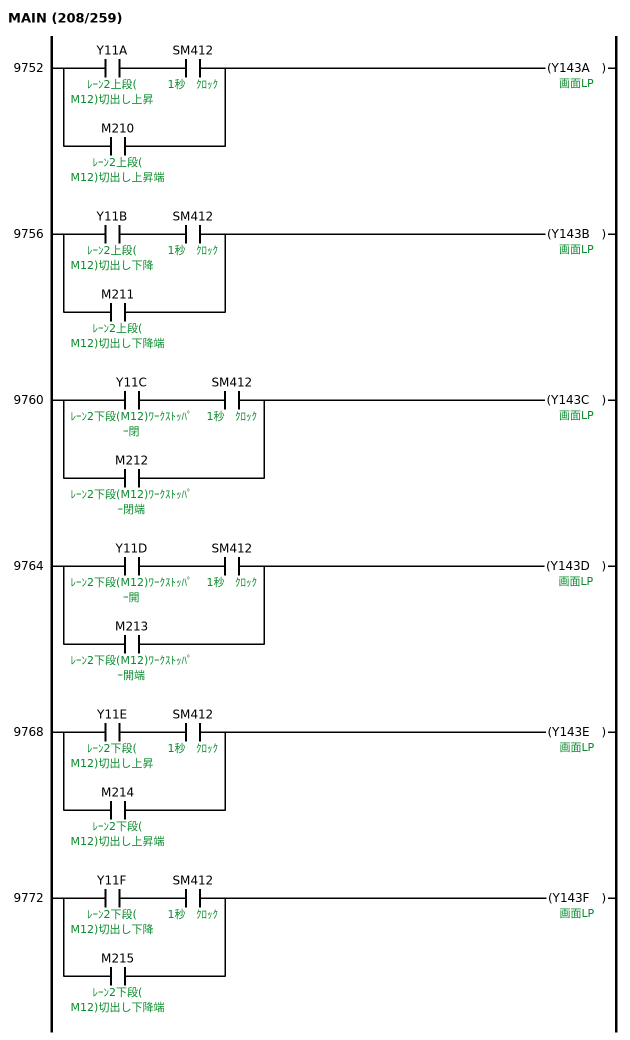
9752  LD      Y11A  ; ﾚｰﾝ2上段(M12)切出し上昇
      AND     SM412  ; 1秒   ｸﾛｯｸ
      OR      M210  ; ﾚｰﾝ2上段(M12)切出し上昇端
      OUT     Y143A  ; 画面LP
9756  LD      Y11B  ; ﾚｰﾝ2上段(M12)切出し下降
      AND     SM412  ; 1秒   ｸﾛｯｸ
      OR      M211  ; ﾚｰﾝ2上段(M12)切出し下降端
      OUT     Y143B  ; 画面LP
9760  LD      Y11C  ; ﾚｰﾝ2下段(M12)ﾜｰｸｽﾄｯﾊﾟｰ閉
      AND     SM412  ; 1秒   ｸﾛｯｸ
      OR      M212  ; ﾚｰﾝ2下段(M12)ﾜｰｸｽﾄｯﾊﾟｰ閉端
      OUT     Y143C  ; 画面LP
9764  LD      Y11D  ; ﾚｰﾝ2下段(M12)ﾜｰｸｽﾄｯﾊﾟｰ開
      AND     SM412  ; 1秒   ｸﾛｯｸ
      OR      M213  ; ﾚｰﾝ2下段(M12)ﾜｰｸｽﾄｯﾊﾟｰ開端
      OUT     Y143D  ; 画面LP
9768  LD      Y11E  ; ﾚｰﾝ2下段(M12)切出し上昇
      AND     SM412  ; 1秒   ｸﾛｯｸ
      OR      M214  ; ﾚｰﾝ2下段(M12)切出し上昇端
      OUT     Y143E  ; 画面LP
9772  LD      Y11F  ; ﾚｰﾝ2下段(M12)切出し下降
      AND     SM412  ; 1秒   ｸﾛｯｸ
      OR      M215  ; ﾚｰﾝ2下段(M12)切出し下降端
      OUT     Y143F  ; 画面LP
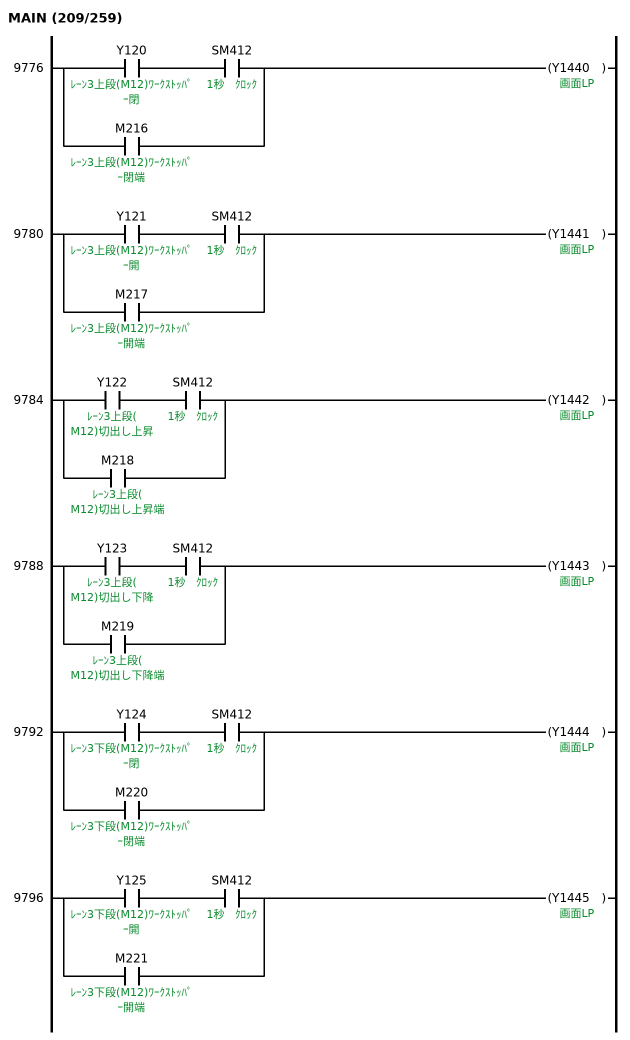
9776  LD      Y120  ; ﾚｰﾝ3上段(M12)ﾜｰｸｽﾄｯﾊﾟｰ閉
      AND     SM412  ; 1秒   ｸﾛｯｸ
      OR      M216  ; ﾚｰﾝ3上段(M12)ﾜｰｸｽﾄｯﾊﾟｰ閉端
      OUT     Y1440  ; 画面LP
9780  LD      Y121  ; ﾚｰﾝ3上段(M12)ﾜｰｸｽﾄｯﾊﾟｰ開
      AND     SM412  ; 1秒   ｸﾛｯｸ
      OR      M217  ; ﾚｰﾝ3上段(M12)ﾜｰｸｽﾄｯﾊﾟｰ開端
      OUT     Y1441  ; 画面LP
9784  LD      Y122  ; ﾚｰﾝ3上段(M12)切出し上昇
      AND     SM412  ; 1秒   ｸﾛｯｸ
      OR      M218  ; ﾚｰﾝ3上段(M12)切出し上昇端
      OUT     Y1442  ; 画面LP
9788  LD      Y123  ; ﾚｰﾝ3上段(M12)切出し下降
      AND     SM412  ; 1秒   ｸﾛｯｸ
      OR      M219  ; ﾚｰﾝ3上段(M12)切出し下降端
      OUT     Y1443  ; 画面LP
9792  LD      Y124  ; ﾚｰﾝ3下段(M12)ﾜｰｸｽﾄｯﾊﾟｰ閉
      AND     SM412  ; 1秒   ｸﾛｯｸ
      OR      M220  ; ﾚｰﾝ3下段(M12)ﾜｰｸｽﾄｯﾊﾟｰ閉端
      OUT     Y1444  ; 画面LP
9796  LD      Y125  ; ﾚｰﾝ3下段(M12)ﾜｰｸｽﾄｯﾊﾟｰ開
      AND     SM412  ; 1秒   ｸﾛｯｸ
      OR      M221  ; ﾚｰﾝ3下段(M12)ﾜｰｸｽﾄｯﾊﾟｰ開端
      OUT     Y1445  ; 画面LP
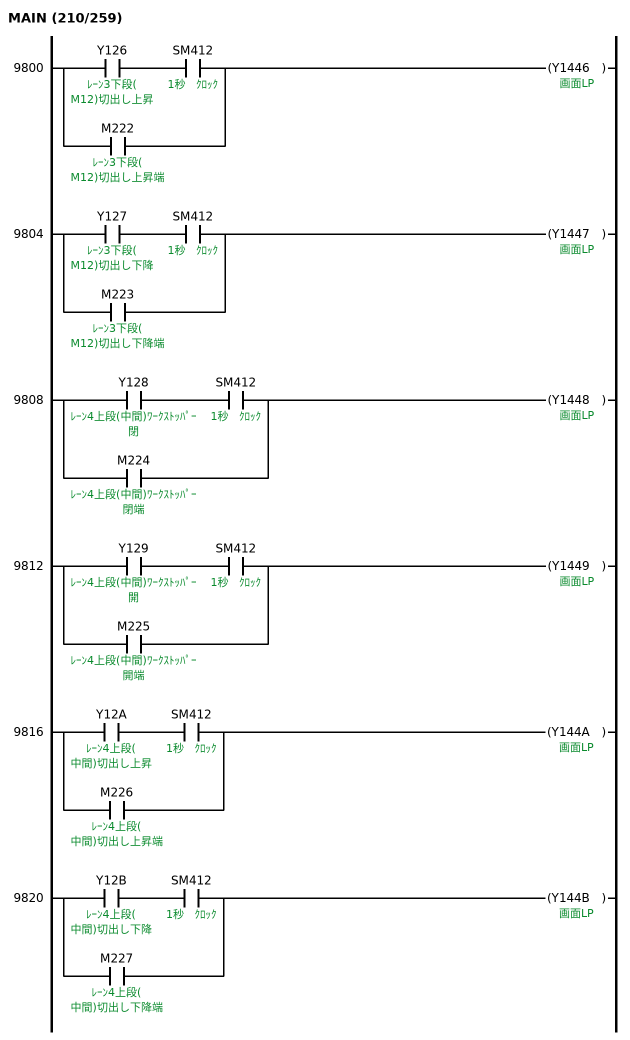
9800  LD      Y126  ; ﾚｰﾝ3下段(M12)切出し上昇
      AND     SM412  ; 1秒   ｸﾛｯｸ
      OR      M222  ; ﾚｰﾝ3下段(M12)切出し上昇端
      OUT     Y1446  ; 画面LP
9804  LD      Y127  ; ﾚｰﾝ3下段(M12)切出し下降
      AND     SM412  ; 1秒   ｸﾛｯｸ
      OR      M223  ; ﾚｰﾝ3下段(M12)切出し下降端
      OUT     Y1447  ; 画面LP
9808  LD      Y128  ; ﾚｰﾝ4上段(中間)ﾜｰｸｽﾄｯﾊﾟｰ閉
      AND     SM412  ; 1秒   ｸﾛｯｸ
      OR      M224  ; ﾚｰﾝ4上段(中間)ﾜｰｸｽﾄｯﾊﾟｰ閉端
      OUT     Y1448  ; 画面LP
9812  LD      Y129  ; ﾚｰﾝ4上段(中間)ﾜｰｸｽﾄｯﾊﾟｰ開
      AND     SM412  ; 1秒   ｸﾛｯｸ
      OR      M225  ; ﾚｰﾝ4上段(中間)ﾜｰｸｽﾄｯﾊﾟｰ開端
      OUT     Y1449  ; 画面LP
9816  LD      Y12A  ; ﾚｰﾝ4上段(中間)切出し上昇
      AND     SM412  ; 1秒   ｸﾛｯｸ
      OR      M226  ; ﾚｰﾝ4上段(中間)切出し上昇端
      OUT     Y144A  ; 画面LP
9820  LD      Y12B  ; ﾚｰﾝ4上段(中間)切出し下降
      AND     SM412  ; 1秒   ｸﾛｯｸ
      OR      M227  ; ﾚｰﾝ4上段(中間)切出し下降端
      OUT     Y144B  ; 画面LP
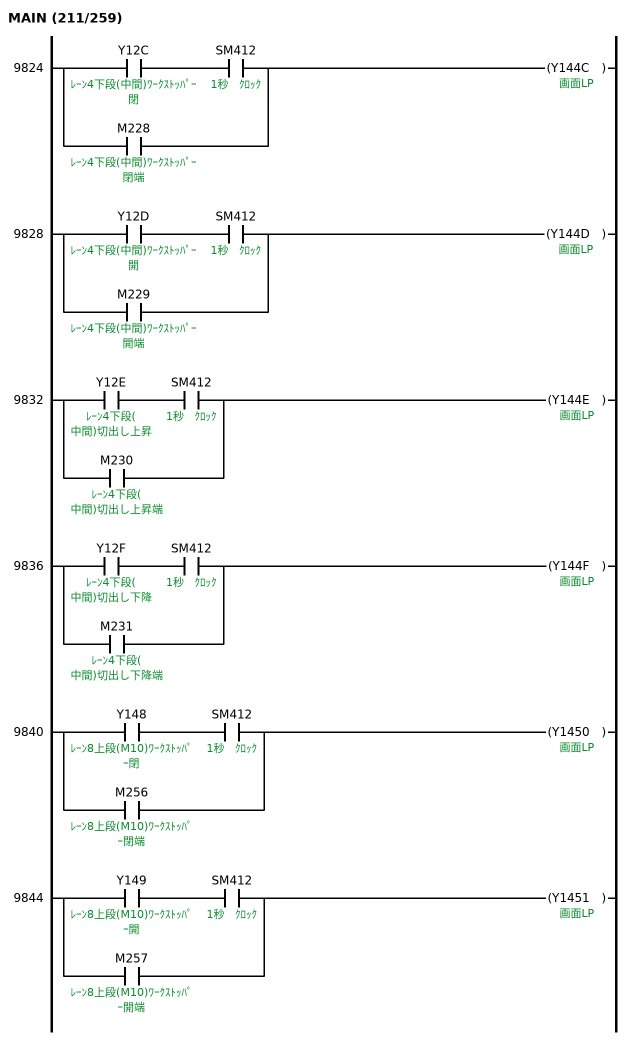
9824  LD      Y12C  ; ﾚｰﾝ4下段(中間)ﾜｰｸｽﾄｯﾊﾟｰ閉
      AND     SM412  ; 1秒   ｸﾛｯｸ
      OR      M228  ; ﾚｰﾝ4下段(中間)ﾜｰｸｽﾄｯﾊﾟｰ閉端
      OUT     Y144C  ; 画面LP
9828  LD      Y12D  ; ﾚｰﾝ4下段(中間)ﾜｰｸｽﾄｯﾊﾟｰ開
      AND     SM412  ; 1秒   ｸﾛｯｸ
      OR      M229  ; ﾚｰﾝ4下段(中間)ﾜｰｸｽﾄｯﾊﾟｰ開端
      OUT     Y144D  ; 画面LP
9832  LD      Y12E  ; ﾚｰﾝ4下段(中間)切出し上昇
      AND     SM412  ; 1秒   ｸﾛｯｸ
      OR      M230  ; ﾚｰﾝ4下段(中間)切出し上昇端
      OUT     Y144E  ; 画面LP
9836  LD      Y12F  ; ﾚｰﾝ4下段(中間)切出し下降
      AND     SM412  ; 1秒   ｸﾛｯｸ
      OR      M231  ; ﾚｰﾝ4下段(中間)切出し下降端
      OUT     Y144F  ; 画面LP
9840  LD      Y148  ; ﾚｰﾝ8上段(M10)ﾜｰｸｽﾄｯﾊﾟｰ閉
      AND     SM412  ; 1秒   ｸﾛｯｸ
      OR      M256  ; ﾚｰﾝ8上段(M10)ﾜｰｸｽﾄｯﾊﾟｰ閉端
      OUT     Y1450  ; 画面LP
9844  LD      Y149  ; ﾚｰﾝ8上段(M10)ﾜｰｸｽﾄｯﾊﾟｰ開
      AND     SM412  ; 1秒   ｸﾛｯｸ
      OR      M257  ; ﾚｰﾝ8上段(M10)ﾜｰｸｽﾄｯﾊﾟｰ開端
      OUT     Y1451  ; 画面LP
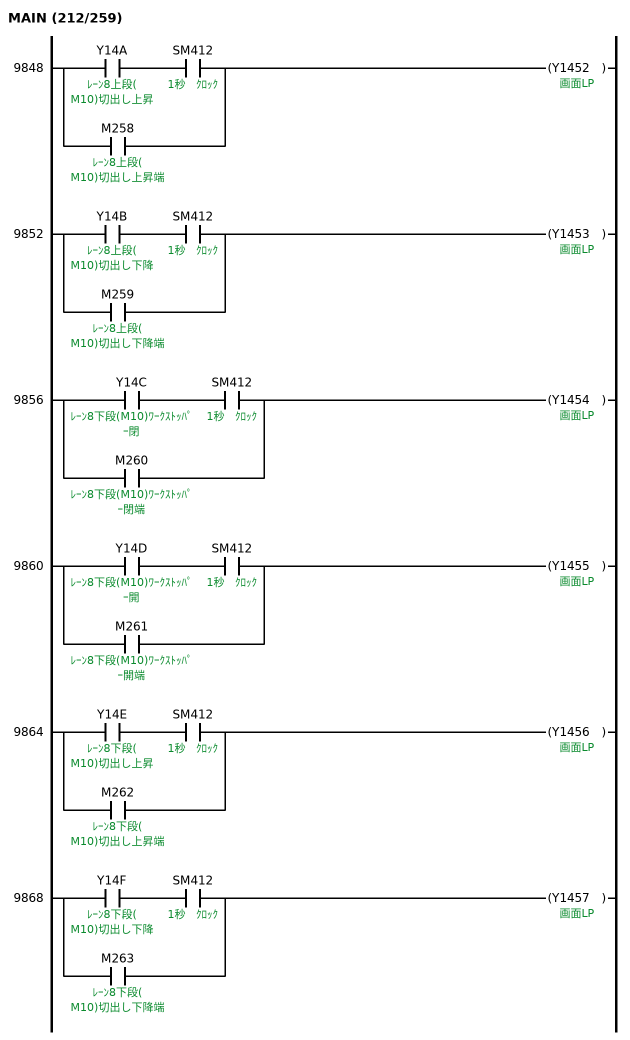
9848  LD      Y14A  ; ﾚｰﾝ8上段(M10)切出し上昇
      AND     SM412  ; 1秒   ｸﾛｯｸ
      OR      M258  ; ﾚｰﾝ8上段(M10)切出し上昇端
      OUT     Y1452  ; 画面LP
9852  LD      Y14B  ; ﾚｰﾝ8上段(M10)切出し下降
      AND     SM412  ; 1秒   ｸﾛｯｸ
      OR      M259  ; ﾚｰﾝ8上段(M10)切出し下降端
      OUT     Y1453  ; 画面LP
9856  LD      Y14C  ; ﾚｰﾝ8下段(M10)ﾜｰｸｽﾄｯﾊﾟｰ閉
      AND     SM412  ; 1秒   ｸﾛｯｸ
      OR      M260  ; ﾚｰﾝ8下段(M10)ﾜｰｸｽﾄｯﾊﾟｰ閉端
      OUT     Y1454  ; 画面LP
9860  LD      Y14D  ; ﾚｰﾝ8下段(M10)ﾜｰｸｽﾄｯﾊﾟｰ開
      AND     SM412  ; 1秒   ｸﾛｯｸ
      OR      M261  ; ﾚｰﾝ8下段(M10)ﾜｰｸｽﾄｯﾊﾟｰ開端
      OUT     Y1455  ; 画面LP
9864  LD      Y14E  ; ﾚｰﾝ8下段(M10)切出し上昇
      AND     SM412  ; 1秒   ｸﾛｯｸ
      OR      M262  ; ﾚｰﾝ8下段(M10)切出し上昇端
      OUT     Y1456  ; 画面LP
9868  LD      Y14F  ; ﾚｰﾝ8下段(M10)切出し下降
      AND     SM412  ; 1秒   ｸﾛｯｸ
      OR      M263  ; ﾚｰﾝ8下段(M10)切出し下降端
      OUT     Y1457  ; 画面LP
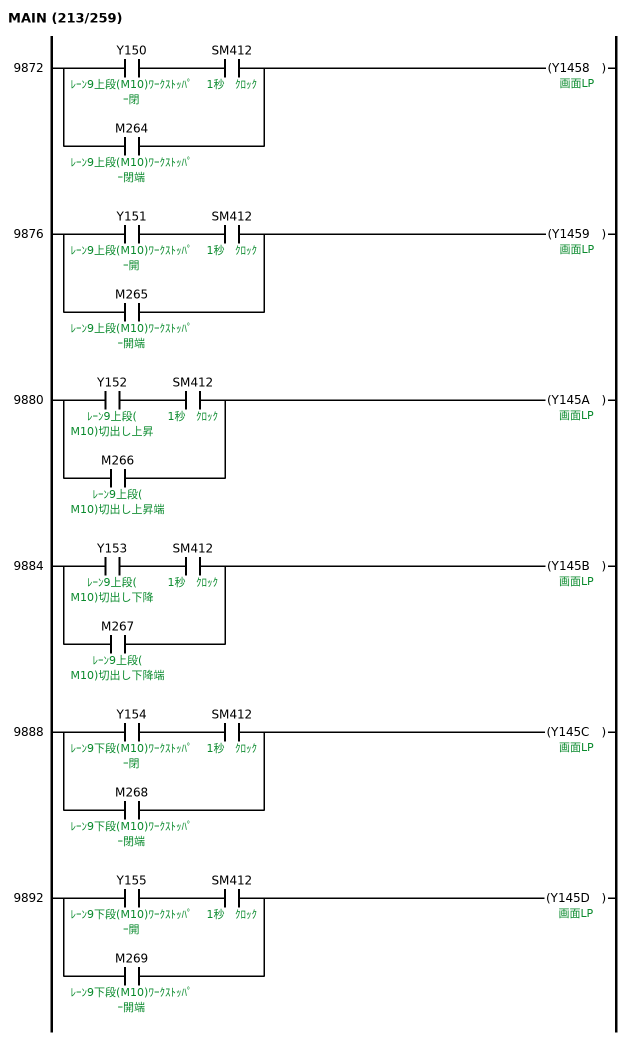
9872  LD      Y150  ; ﾚｰﾝ9上段(M10)ﾜｰｸｽﾄｯﾊﾟｰ閉
      AND     SM412  ; 1秒   ｸﾛｯｸ
      OR      M264  ; ﾚｰﾝ9上段(M10)ﾜｰｸｽﾄｯﾊﾟｰ閉端
      OUT     Y1458  ; 画面LP
9876  LD      Y151  ; ﾚｰﾝ9上段(M10)ﾜｰｸｽﾄｯﾊﾟｰ開
      AND     SM412  ; 1秒   ｸﾛｯｸ
      OR      M265  ; ﾚｰﾝ9上段(M10)ﾜｰｸｽﾄｯﾊﾟｰ開端
      OUT     Y1459  ; 画面LP
9880  LD      Y152  ; ﾚｰﾝ9上段(M10)切出し上昇
      AND     SM412  ; 1秒   ｸﾛｯｸ
      OR      M266  ; ﾚｰﾝ9上段(M10)切出し上昇端
      OUT     Y145A  ; 画面LP
9884  LD      Y153  ; ﾚｰﾝ9上段(M10)切出し下降
      AND     SM412  ; 1秒   ｸﾛｯｸ
      OR      M267  ; ﾚｰﾝ9上段(M10)切出し下降端
      OUT     Y145B  ; 画面LP
9888  LD      Y154  ; ﾚｰﾝ9下段(M10)ﾜｰｸｽﾄｯﾊﾟｰ閉
      AND     SM412  ; 1秒   ｸﾛｯｸ
      OR      M268  ; ﾚｰﾝ9下段(M10)ﾜｰｸｽﾄｯﾊﾟｰ閉端
      OUT     Y145C  ; 画面LP
9892  LD      Y155  ; ﾚｰﾝ9下段(M10)ﾜｰｸｽﾄｯﾊﾟｰ開
      AND     SM412  ; 1秒   ｸﾛｯｸ
      OR      M269  ; ﾚｰﾝ9下段(M10)ﾜｰｸｽﾄｯﾊﾟｰ開端
      OUT     Y145D  ; 画面LP
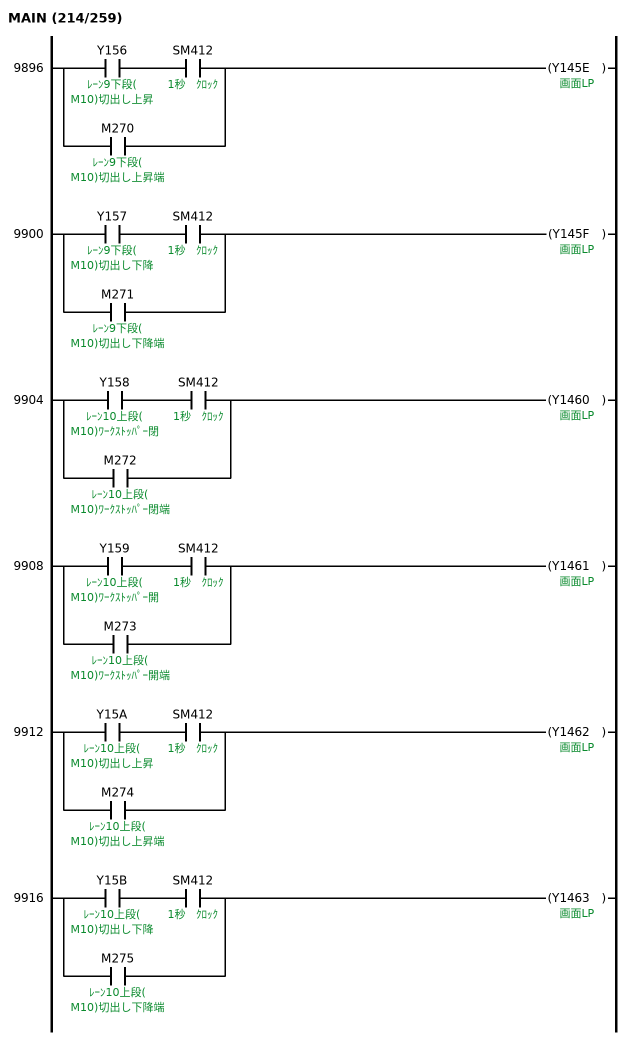
9896  LD      Y156  ; ﾚｰﾝ9下段(M10)切出し上昇
      AND     SM412  ; 1秒   ｸﾛｯｸ
      OR      M270  ; ﾚｰﾝ9下段(M10)切出し上昇端
      OUT     Y145E  ; 画面LP
9900  LD      Y157  ; ﾚｰﾝ9下段(M10)切出し下降
      AND     SM412  ; 1秒   ｸﾛｯｸ
      OR      M271  ; ﾚｰﾝ9下段(M10)切出し下降端
      OUT     Y145F  ; 画面LP
9904  LD      Y158  ; ﾚｰﾝ10上段(M10)ﾜｰｸｽﾄｯﾊﾟｰ閉
      AND     SM412  ; 1秒   ｸﾛｯｸ
      OR      M272  ; ﾚｰﾝ10上段(M10)ﾜｰｸｽﾄｯﾊﾟｰ閉端
      OUT     Y1460  ; 画面LP
9908  LD      Y159  ; ﾚｰﾝ10上段(M10)ﾜｰｸｽﾄｯﾊﾟｰ開
      AND     SM412  ; 1秒   ｸﾛｯｸ
      OR      M273  ; ﾚｰﾝ10上段(M10)ﾜｰｸｽﾄｯﾊﾟｰ開端
      OUT     Y1461  ; 画面LP
9912  LD      Y15A  ; ﾚｰﾝ10上段(M10)切出し上昇
      AND     SM412  ; 1秒   ｸﾛｯｸ
      OR      M274  ; ﾚｰﾝ10上段(M10)切出し上昇端
      OUT     Y1462  ; 画面LP
9916  LD      Y15B  ; ﾚｰﾝ10上段(M10)切出し下降
      AND     SM412  ; 1秒   ｸﾛｯｸ
      OR      M275  ; ﾚｰﾝ10上段(M10)切出し下降端
      OUT     Y1463  ; 画面LP
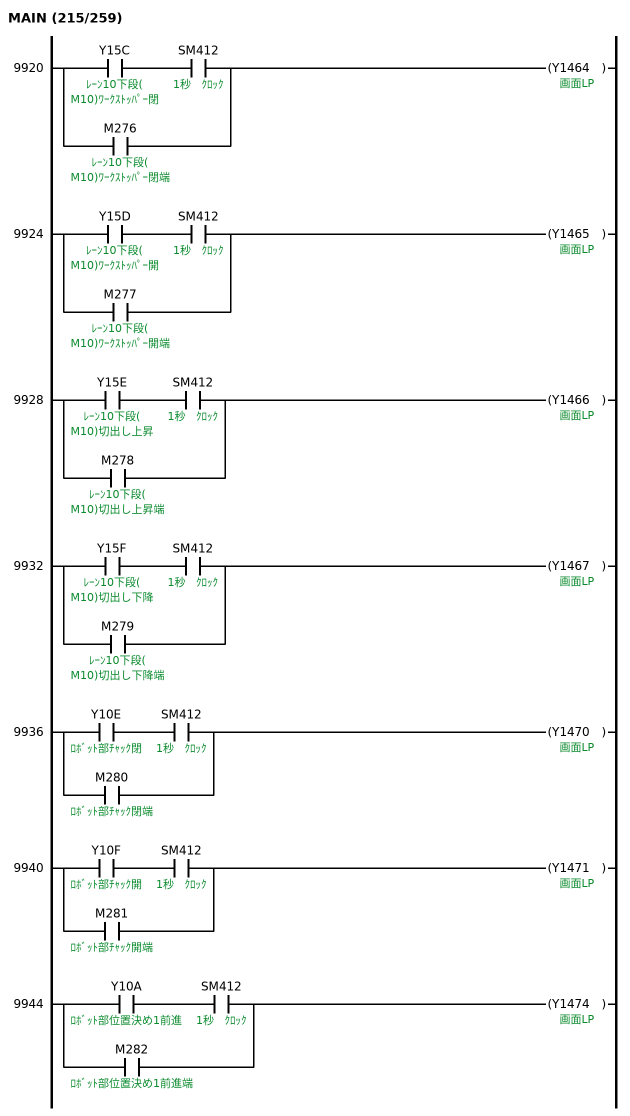
9920  LD      Y15C  ; ﾚｰﾝ10下段(M10)ﾜｰｸｽﾄｯﾊﾟｰ閉
      AND     SM412  ; 1秒   ｸﾛｯｸ
      OR      M276  ; ﾚｰﾝ10下段(M10)ﾜｰｸｽﾄｯﾊﾟｰ閉端
      OUT     Y1464  ; 画面LP
9924  LD      Y15D  ; ﾚｰﾝ10下段(M10)ﾜｰｸｽﾄｯﾊﾟｰ開
      AND     SM412  ; 1秒   ｸﾛｯｸ
      OR      M277  ; ﾚｰﾝ10下段(M10)ﾜｰｸｽﾄｯﾊﾟｰ開端
      OUT     Y1465  ; 画面LP
9928  LD      Y15E  ; ﾚｰﾝ10下段(M10)切出し上昇
      AND     SM412  ; 1秒   ｸﾛｯｸ
      OR      M278  ; ﾚｰﾝ10下段(M10)切出し上昇端
      OUT     Y1466  ; 画面LP
9932  LD      Y15F  ; ﾚｰﾝ10下段(M10)切出し下降
      AND     SM412  ; 1秒   ｸﾛｯｸ
      OR      M279  ; ﾚｰﾝ10下段(M10)切出し下降端
      OUT     Y1467  ; 画面LP
9936  LD      Y10E  ; ﾛﾎﾞｯﾄ部ﾁｬｯｸ閉
      AND     SM412  ; 1秒   ｸﾛｯｸ
      OR      M280  ; ﾛﾎﾞｯﾄ部ﾁｬｯｸ閉端
      OUT     Y1470  ; 画面LP
9940  LD      Y10F  ; ﾛﾎﾞｯﾄ部ﾁｬｯｸ開
      AND     SM412  ; 1秒   ｸﾛｯｸ
      OR      M281  ; ﾛﾎﾞｯﾄ部ﾁｬｯｸ開端
      OUT     Y1471  ; 画面LP
9944  LD      Y10A  ; ﾛﾎﾞｯﾄ部位置決め1前進
      AND     SM412  ; 1秒   ｸﾛｯｸ
      OR      M282  ; ﾛﾎﾞｯﾄ部位置決め1前進端
      OUT     Y1474  ; 画面LP
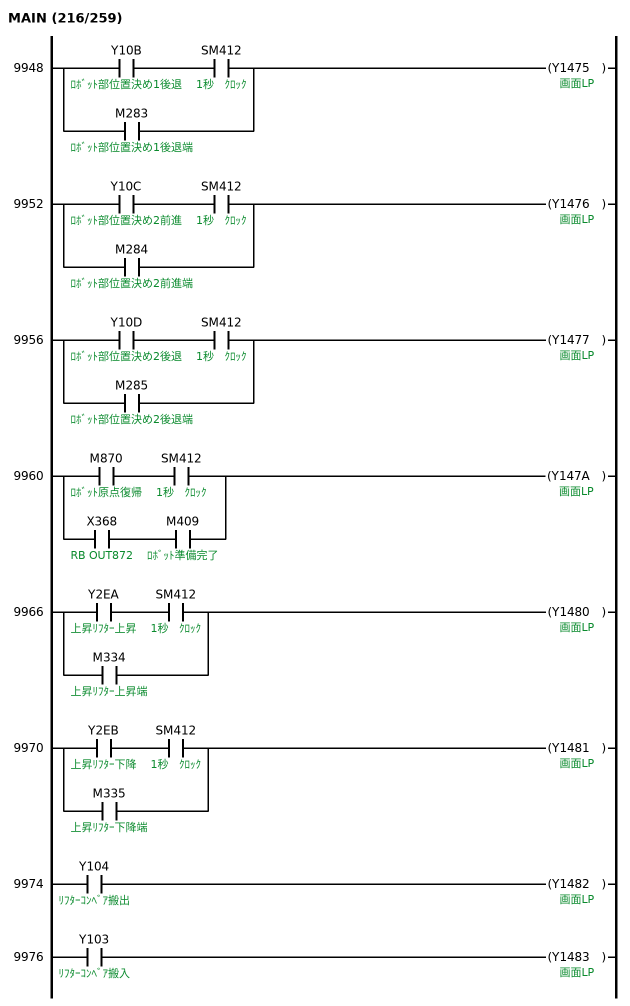
9948  LD      Y10B  ; ﾛﾎﾞｯﾄ部位置決め1後退
      AND     SM412  ; 1秒   ｸﾛｯｸ
      OR      M283  ; ﾛﾎﾞｯﾄ部位置決め1後退端
      OUT     Y1475  ; 画面LP
9952  LD      Y10C  ; ﾛﾎﾞｯﾄ部位置決め2前進
      AND     SM412  ; 1秒   ｸﾛｯｸ
      OR      M284  ; ﾛﾎﾞｯﾄ部位置決め2前進端
      OUT     Y1476  ; 画面LP
9956  LD      Y10D  ; ﾛﾎﾞｯﾄ部位置決め2後退
      AND     SM412  ; 1秒   ｸﾛｯｸ
      OR      M285  ; ﾛﾎﾞｯﾄ部位置決め2後退端
      OUT     Y1477  ; 画面LP
9960  LD      M870  ; ﾛﾎﾞｯﾄ原点復帰
      AND     SM412  ; 1秒   ｸﾛｯｸ
      LD      X368  ; RB OUT872
      AND     M409  ; ﾛﾎﾞｯﾄ準備完了
      ORB
      OUT     Y147A  ; 画面LP
9966  LD      Y2EA  ; 上昇ﾘﾌﾀｰ上昇
      AND     SM412  ; 1秒   ｸﾛｯｸ
      OR      M334  ; 上昇ﾘﾌﾀｰ上昇端
      OUT     Y1480  ; 画面LP
9970  LD      Y2EB  ; 上昇ﾘﾌﾀｰ下降
      AND     SM412  ; 1秒   ｸﾛｯｸ
      OR      M335  ; 上昇ﾘﾌﾀｰ下降端
      OUT     Y1481  ; 画面LP
9974  LD      Y104  ; ﾘﾌﾀｰｺﾝﾍﾞｱ搬出
      OUT     Y1482  ; 画面LP
9976  LD      Y103  ; ﾘﾌﾀｰｺﾝﾍﾞｱ搬入
      OUT     Y1483  ; 画面LP
